Staubli VAL3: listEmpty.pgx

public program listEmpty()
  local num i
  local num l_nSize
begin
  //-----------------------------------------------------------------------
  //Header begin
  //Description of program
  //  Delete all the elements of the list (sItems).
  //  删除列表（sItems）中的所有元素
  //Example
  //  call listEmpty()
  //
  //History
  //  Creation : 28-04-08 - f.Rob
  //Header end
  //-----------------------------------------------------------------------
  l_nSize=size(sItems)-1
  for i=0 to l_nSize
    if i>0
      //Destroy all elements of sItems 删除sItems中的所有元素
      delete(sItems[0])
      //Destroy all elements of bReadWrite  删除bReadWrite中的所有元素
      delete(bReadWrite[0])
    endIf
  endFor
  sItems=""
end
